TYPE DAQ_CTR :
STRUCT
	//clears all data from data arrays
	CMDDATACLR		:BOOL;
	//controls whether data is appended to current file or not
	CMDDATAAPEND	:BOOL;
	CMDDATAWRITE	:BOOL;
	CMDCSVRESET		:BOOL;
	CMDSICKPROFILE	:BOOL;
	DAQRES			:INT := 1; //acquire every x mm or seconds (default 1)
END_STRUCT
END_TYPE

(* stored: Version 1.1.0.1, ProductVersion 3.1.4026.12
   DUT DAQ_CTR: Id {9bc06f9c-a6c9-47ae-966a-864e0de7397d} *)
